INTERFACE ITF_SaMControllerCommandChange

METHOD PUBLIC ChangeModeTo
VAR_INPUT
	eNewMode			: E_BaseMachineMode;
END_VAR
END_METHOD

METHOD PUBLIC ChangeStateTo
VAR_INPUT
	eNewState			: E_BaseMachineState;
END_VAR
END_METHOD

METHOD PUBLIC GetState : E_BaseMachineState
VAR_INPUT
END_VAR
END_METHOD

METHOD IsModeEnebles : BOOL
VAR_INPUT
	eMode			: E_BaseMachineMode;
END_VAR
END_METHOD

METHOD IsPossibleExitActiveState : BOOL
VAR_INPUT
END_VAR
END_METHOD

METHOD IsPossibleExitState : BOOL
VAR_INPUT
	eMode		: E_BaseMachineMode;
END_VAR
END_METHOD

METHOD PUBLIC IsStateInModeEnabled : BOOL
VAR_INPUT
	eState			: E_BaseMachineState;
END_VAR
END_METHOD

END_INTERFACE

(* stored: Version 1.1.0.1
   Itf ITF_SaMControllerCommandChange: Id {4f3c20a9-bad8-0c25-32a4-4d92805aad72}
   Method ChangeModeTo: Id {438f8f9d-6699-052d-3a6f-112ca53c6c0f}
   Method ChangeStateTo: Id {20e110f3-d687-003b-0708-468cc54e6e0f}
   Method GetState: Id {2d9fe36b-32c7-049a-021e-6cda6bb4eaab}
   Method IsModeEnebles: Id {6a423769-8c8d-07e3-138a-e7ec7acacb3e}
   Method IsPossibleExitActiveState: Id {653e7c6d-6acc-090e-2947-56adaa34f221}
   Method IsPossibleExitState: Id {41333180-94d8-0463-3725-199c7f48084c}
   Method IsStateInModeEnabled: Id {8b94b531-de78-0248-28cf-4d8a71b21e15} *)
